(****************************************************************************************)
(*							Beckhoff Automation Poland									*)
(*								F_2Bytes_To_Word v1.0									*)
(*									15.02.2010											*)
(*		Funkcja tworząca zmienną typu WORD z dwóch zmiennych typu BYTE					*)
(*______________________________________________________________________________________*)
FUNCTION F_2Bytes_To_Word : WORD
VAR_INPUT
	byHigh	:	BYTE;
	byLow	:	BYTE;
END_VAR
VAR
END_VAR

F_2Bytes_To_Word := byHigh;
F_2Bytes_To_Word := SHL(F_2Bytes_To_Word,8);
F_2Bytes_To_Word := F_2Bytes_To_Word + byLow;

END_FUNCTION

(* stored: Version 1.1.0.1, ProductVersion 3.1.4026.13, FileIdentifier 9fd695d57e079b5faf4d42a48450b07fac8c0732, FileSignature 74728dfa76211c2b26eb768cac9ecd5b96d5f35fd8794d656ec87008a50d04dd36bcfc5e7259ff8ed62271cb7623f6ad8b45a89b419fd57f7735a5c175361ed7cc85a4317c654a911041aa03efe7c9fd8f6848f2f038fc7aebe692303daec2d731eef565e6b54db0f13f68df3b91b9461e03ae03179f2fd21e0c9bb346368e3294ffbe14d8e8f6d960c9f5a071e8fb5ba56e96786076a3370c88e28ee403e229fe621e56e2e4c2e16ff53bad91d8812c94b766e06711b3f54c0e8a95dd662847c7797305dbe3e036290b827a7bd2ec4d6bd785d2924f3229bedd52f93c8bd2ab38fd5eaa734bd51fb71970728996623b2d7035b2a17ebd1a2ed244f849e2ae65
   POU F_2Bytes_To_Word: Id {0bcfedca-596a-4772-a3fc-9abcd797c20f}, SpecialFunc None *)
